FUNCTION_BLOCK AtvResetErrorLogic (* Basic Function Block Type *)
  (* Standard: 61499-2 *)
  (* Version 0.1, 10/6/2026, SESA713705, Schneider Electric, Hidryco 10/2026: reset automatico limitado a 3 tentativas por ocorrencia (antes era infinito 3 s / 1 s); depois so pela IHM ou em nova ocorrencia *)
  PACKAGE SE.Nereda;
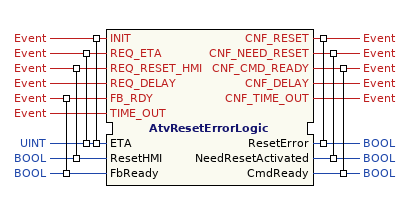
  EVENT_INPUT
    INIT WITH ETA; (* Initialization Request *)
    REQ_ETA WITH ETA; (* Normal Execution Request *)
    REQ_RESET_HMI WITH ResetHMI;
    REQ_DELAY;
    FB_RDY WITH FbReady;
    TIME_OUT;
  END_EVENT
  EVENT_OUTPUT
    CNF_RESET WITH ResetError; (* Execution Confirmation *)
    CNF_NEED_RESET WITH NeedResetActivated;
    CNF_CMD_READY WITH CmdReady;
    CNF_DELAY;
    CNF_TIME_OUT;
  END_EVENT
  VAR_INPUT
    ETA : UINT;
    ResetHMI : BOOL;
    FbReady : BOOL;
  END_VAR
  VAR_OUTPUT
    ResetError : BOOL;
    NeedResetActivated : BOOL;
    CmdReady : BOOL;
  END_VAR
  VAR
    Tries : INT := 0; (* Tentativas de reset automatico na ocorrencia atual *)
  END_VAR
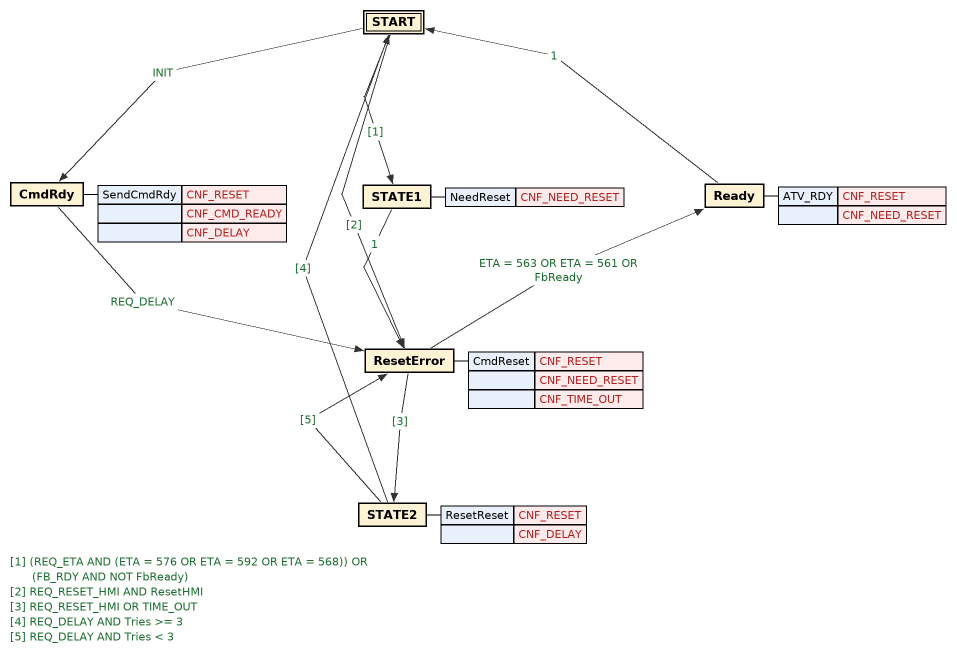
  EC_STATES
    START; (* Initial State *)
    Ready : ATV_RDY -> CNF_RESET, -> CNF_NEED_RESET;
    CmdRdy : SendCmdRdy -> CNF_RESET, -> CNF_CMD_READY, -> CNF_DELAY;
    ResetError : CmdReset -> CNF_RESET, -> CNF_NEED_RESET, -> CNF_TIME_OUT;
    STATE1 : NeedReset -> CNF_NEED_RESET;
    STATE2 : ResetReset -> CNF_RESET, -> CNF_DELAY;
  END_STATES
  EC_TRANSITIONS
    START TO CmdRdy := INIT;
    CmdRdy TO ResetError := REQ_DELAY;
    ResetError TO Ready := ETA = 563 OR ETA = 561 OR FbReady;
    Ready TO START := 1;
    START TO STATE1 := (REQ_ETA AND (ETA = 576 OR ETA = 592 OR ETA = 568)) OR (FB_RDY AND NOT FbReady);
    STATE1 TO ResetError := 1;
    ResetError TO STATE2 := REQ_RESET_HMI OR TIME_OUT;
    STATE2 TO ResetError := REQ_DELAY AND Tries < 3;
    STATE2 TO START := REQ_DELAY AND Tries >= 3;
    START TO ResetError := REQ_RESET_HMI AND ResetHMI;
  END_TRANSITIONS
  ALGORITHM INIT IN ST: (* Initialization algorithm *)
;
ResetError := FALSE;
CmdReady := TRUE;
  END_ALGORITHM
  ALGORITHM ATV_RDY IN ST:
;
ResetError := FALSE;
NeedResetActivated := FALSE;
Tries := 0;
  END_ALGORITHM
  ALGORITHM NeedReset IN ST:
;
NeedResetActivated := TRUE;
Tries := 0;
  END_ALGORITHM
  ALGORITHM CmdReset IN ST:
ResetError := TRUE;
NeedResetActivated := TRUE;
Tries := Tries + 1;
  END_ALGORITHM
  ALGORITHM SendCmdRdy IN ST:
ResetError := FALSE;
CmdReady := TRUE;
  END_ALGORITHM
  ALGORITHM SensResetHMI IN ST:
;
ResetError := ResetHMI;
  END_ALGORITHM
  ALGORITHM ResetReset IN ST:
;
ResetError := FALSE;
  END_ALGORITHM
END_FUNCTION_BLOCK
